// TIA Portal V19 export
TYPE "DecoilersHRot_Manager"
   STRUCT
      EnableStopDoorOpeningReq : Bool;
      EnableStopInPhase : Bool;
      EnableStopProgrammed : Bool;
      Control_ON : Bool;
      Decoiler1_MoveInLine : Bool;
      Decoiler2_MoveInLine : Bool;
      ChangeDecoilerEnable : Bool;
   END_STRUCT;
END_TYPE
